VAR_GLOBAL // INPUTS
    ivar_inp AT %I*: LREAL;
END_VAR

(* stored: ProductVersion 3.1.0.18, Version 1.1.0.1 *)
